// Mitsubishi GX Works2 project: 타이머응용4   PLC: Q02/Q02H

PROGRAM MAIN
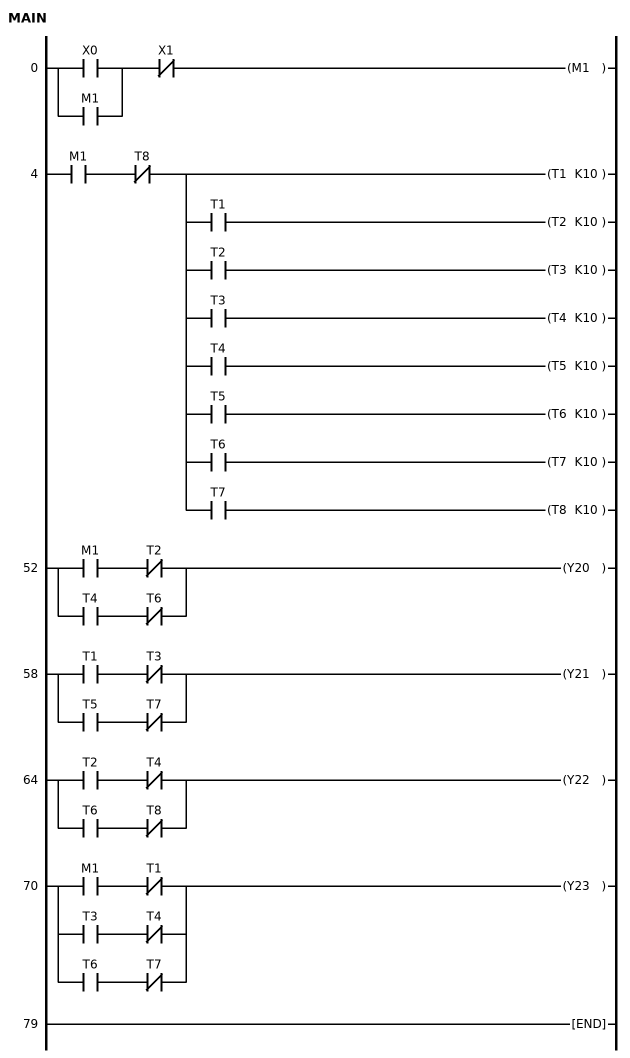
0     LD      X0
      OR      M1
      ANI     X1
      OUT     M1
4     LD      M1
      ANI     T8
      OUT     T1 K10
      MPS
      AND     T1
      OUT     T2 K10
      MRD
      AND     T2
      OUT     T3 K10
      MRD
      AND     T3
      OUT     T4 K10
      MRD
      AND     T4
      OUT     T5 K10
      MRD
      AND     T5
      OUT     T6 K10
      MRD
      AND     T6
      OUT     T7 K10
      MPP
      AND     T7
      OUT     T8 K10
52    LD      M1
      ANI     T2
      LD      T4
      ANI     T6
      ORB
      OUT     Y20
58    LD      T1
      ANI     T3
      LD      T5
      ANI     T7
      ORB
      OUT     Y21
64    LD      T2
      ANI     T4
      LD      T6
      ANI     T8
      ORB
      OUT     Y22
70    LD      M1
      ANI     T1
      LD      T3
      ANI     T4
      ORB
      LD      T6
      ANI     T7
      ORB
      OUT     Y23
79    END
END_PROGRAM
